FUNCTION QUARTERS_TO_LWORD
  (* Standard: 61499-1 *)
  (* Version 1.0, 2024-02-22, franz *)
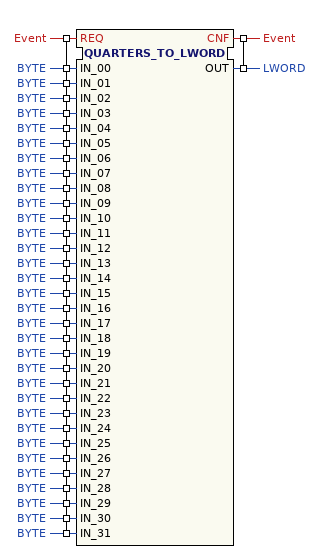
  EVENT_INPUT
    REQ WITH IN_00, IN_01, IN_02, IN_03, IN_04, IN_05, IN_06, IN_07, IN_08, IN_09, IN_10, IN_11, IN_12, IN_13, IN_14, IN_15, IN_16, IN_17, IN_18, IN_19, IN_20, IN_21, IN_22, IN_23, IN_24, IN_25, IN_26, IN_27, IN_28, IN_29, IN_30, IN_31; (* Normal Execution Request *)
  END_EVENT
  EVENT_OUTPUT
    CNF WITH OUT; (* Execution Confirmation *)
  END_EVENT
  VAR_INPUT
    IN_00 : BYTE; (* QUARTER BYTE 00 *)
    IN_01 : BYTE; (* QUARTER BYTE 01 *)
    IN_02 : BYTE; (* QUARTER BYTE 02 *)
    IN_03 : BYTE; (* QUARTER BYTE 03 *)
    IN_04 : BYTE; (* QUARTER BYTE 04 *)
    IN_05 : BYTE; (* QUARTER BYTE 05 *)
    IN_06 : BYTE; (* QUARTER BYTE 06 *)
    IN_07 : BYTE; (* QUARTER BYTE 07 *)
    IN_08 : BYTE; (* QUARTER BYTE 08 *)
    IN_09 : BYTE; (* QUARTER BYTE 09 *)
    IN_10 : BYTE; (* QUARTER BYTE 10 *)
    IN_11 : BYTE; (* QUARTER BYTE 11 *)
    IN_12 : BYTE; (* QUARTER BYTE 12 *)
    IN_13 : BYTE; (* QUARTER BYTE 13 *)
    IN_14 : BYTE; (* QUARTER BYTE 14 *)
    IN_15 : BYTE; (* QUARTER BYTE 15 *)
    IN_16 : BYTE; (* QUARTER BYTE 16 *)
    IN_17 : BYTE; (* QUARTER BYTE 17 *)
    IN_18 : BYTE; (* QUARTER BYTE 18 *)
    IN_19 : BYTE; (* QUARTER BYTE 19 *)
    IN_20 : BYTE; (* QUARTER BYTE 20 *)
    IN_21 : BYTE; (* QUARTER BYTE 21 *)
    IN_22 : BYTE; (* QUARTER BYTE 22 *)
    IN_23 : BYTE; (* QUARTER BYTE 23 *)
    IN_24 : BYTE; (* QUARTER BYTE 24 *)
    IN_25 : BYTE; (* QUARTER BYTE 25 *)
    IN_26 : BYTE; (* QUARTER BYTE 26 *)
    IN_27 : BYTE; (* QUARTER BYTE 27 *)
    IN_28 : BYTE; (* QUARTER BYTE 28 *)
    IN_29 : BYTE; (* QUARTER BYTE 29 *)
    IN_30 : BYTE; (* QUARTER BYTE 30 *)
    IN_31 : BYTE; (* QUARTER BYTE 31 *)
  END_VAR
  VAR_OUTPUT
    OUT : LWORD; (* LWORD Output *)
  END_VAR
  BODY IN ST:
FUNCTION QUARTERS_TO_LWORD

VAR_INPUT
	IN_00 : BYTE;    // QUARTER BYTE 00
	IN_01 : BYTE;    // QUARTER BYTE 01
	IN_02 : BYTE;    // QUARTER BYTE 02
	IN_03 : BYTE;    // QUARTER BYTE 03
	IN_04 : BYTE;    // QUARTER BYTE 04
	IN_05 : BYTE;    // QUARTER BYTE 05
	IN_06 : BYTE;    // QUARTER BYTE 06
	IN_07 : BYTE;    // QUARTER BYTE 07
	IN_08 : BYTE;    // QUARTER BYTE 08
	IN_09 : BYTE;    // QUARTER BYTE 09
	IN_10 : BYTE;    // QUARTER BYTE 10
	IN_11 : BYTE;    // QUARTER BYTE 11
	IN_12 : BYTE;    // QUARTER BYTE 12
	IN_13 : BYTE;    // QUARTER BYTE 13
	IN_14 : BYTE;    // QUARTER BYTE 14
	IN_15 : BYTE;    // QUARTER BYTE 15
	IN_16 : BYTE;    // QUARTER BYTE 16
	IN_17 : BYTE;    // QUARTER BYTE 17
	IN_18 : BYTE;    // QUARTER BYTE 18
	IN_19 : BYTE;    // QUARTER BYTE 19
	IN_20 : BYTE;    // QUARTER BYTE 20
	IN_21 : BYTE;    // QUARTER BYTE 21
	IN_22 : BYTE;    // QUARTER BYTE 22
	IN_23 : BYTE;    // QUARTER BYTE 23
	IN_24 : BYTE;    // QUARTER BYTE 24
	IN_25 : BYTE;    // QUARTER BYTE 25
	IN_26 : BYTE;    // QUARTER BYTE 26
	IN_27 : BYTE;    // QUARTER BYTE 27
	IN_28 : BYTE;    // QUARTER BYTE 28
	IN_29 : BYTE;    // QUARTER BYTE 29
	IN_30 : BYTE;    // QUARTER BYTE 30
	IN_31 : BYTE;    // QUARTER BYTE 31
END_VAR

VAR_OUTPUT
	OUT : LWORD;    // LWORD Output
END_VAR

(* this Function combines the 31 QUARTER BYTES to a lword *)
OUT := SHL(IN_31, SHIFT_QUARTER_31)
	OR SHL(IN_30, SHIFT_QUARTER_30)
	OR SHL(IN_29, SHIFT_QUARTER_29)
	OR SHL(IN_28, SHIFT_QUARTER_28)
	OR SHL(IN_27, SHIFT_QUARTER_27)
	OR SHL(IN_26, SHIFT_QUARTER_26)
	OR SHL(IN_25, SHIFT_QUARTER_25)
	OR SHL(IN_24, SHIFT_QUARTER_24)
	OR SHL(IN_23, SHIFT_QUARTER_23)
	OR SHL(IN_22, SHIFT_QUARTER_22)
	OR SHL(IN_21, SHIFT_QUARTER_21)
	OR SHL(IN_20, SHIFT_QUARTER_20)
	OR SHL(IN_19, SHIFT_QUARTER_19)
	OR SHL(IN_18, SHIFT_QUARTER_18)
	OR SHL(IN_17, SHIFT_QUARTER_17)
	OR SHL(IN_16, SHIFT_QUARTER_16)
	OR SHL(IN_15, SHIFT_QUARTER_15)
	OR SHL(IN_14, SHIFT_QUARTER_14)
	OR SHL(IN_13, SHIFT_QUARTER_13)
	OR SHL(IN_12, SHIFT_QUARTER_12)
	OR SHL(IN_11, SHIFT_QUARTER_11)
	OR SHL(IN_10, SHIFT_QUARTER_10)
	OR SHL(IN_09, SHIFT_QUARTER_09)
	OR SHL(IN_08, SHIFT_QUARTER_08)
	OR SHL(IN_07, SHFT_QUARTER_07)
	OR SHL(IN_06, SHFT_QUARTER_06)
	OR SHL(IN_05, SHFT_QUARTER_05)
	OR SHL(IN_04, SHFT_QUARTER_04)
	OR SHL(IN_03, SHFT_QUARTER_03)
	OR SHL(IN_02, SHFT_QUARTER_02)
	OR SHL(IN_01, SHFT_QUARTER_01)
	OR SHL(IN_00, SHFT_QUARTER_00);

END_FUNCTION
  END_BODY
END_FUNCTION
